{attribute 'GeneratedUsingTerminal: EL3201-0000-0016'}
{attribute addProperty BoxType "EL3201-0000-0016"}
{attribute addProperty Id "EtcSlaveTerminalBaseRTD_InputsAT %I*RTD_Inputs_EA9DF21E9WcStateAT %I*WcState_9091E0EB2InfoDataAT %I*InfoData_32EB74EA10"}
{attribute addProperty CRC "2801983511"}
{attribute addProperty Size "21"}
TYPE EL3201_A702E017 EXTENDS EtcSlaveTerminalBase :
STRUCT
	{attribute addProperty Name "RTD_Inputs"}
	RTD_Inputs : RTD_Inputs_EA9DF21E;
	{attribute addProperty Name "WcState"}
	WcState : WcState_9091E0EB;
	{attribute addProperty Name "InfoData"}
	InfoData : InfoData_32EB74EA;
END_STRUCT
END_TYPE

(* stored: Version 1.2.0.0, ProductVersion 3.1.4024.9
   DUT EL3201_A702E017: Id {1fa22675-7f97-4b6c-bcc6-d145537f0e9e} *)
